FUNCTION_BLOCK FB_Normalize
VAR_INPUT
	nRawInput : INT;
	fMaxValue : LREAL;
END_VAR
VAR_OUTPUT
	fNormalizedInput : LREAL;
END_VAR
VAR
END_VAR

fNormalizedInput := (fMaxValue	* INT_TO_LREAL(nRawInput)) / 32767.0;

fNormalizedInput := LIMIT(0, fNormalizedInput, fMaxValue);

END_FUNCTION_BLOCK

(* stored: Version 1.1.0.1
   POU FB_Normalize: Id {1cb17eff-b342-48b7-ab9a-2d7d641deba9}, SpecialFunc None *)
